{attribute 'GeneratedUsingTerminal: EL5112-0000-0016'}
{attribute addProperty BoxType "EL5112-0000-0016"}
{attribute addProperty Description "EL5112 2Ch. Inc. Encoder 5V (2xAB or 1xABC RS422,TTL)"}
{attribute addProperty Physics "KK"}
{attribute addProperty Id "ENC_Status_Channel_1AT %I*ENC_Status_Channel_10A67E5232ENC_Control_Channel_1AT %Q*ENC_Control_Channel_4C8A739514WcStateAT %I*WcState_9091E0EB2InfoDataAT %I*InfoData_32EB74EA10"}
{attribute addProperty CRC "2247317062"}
{attribute addProperty Size "58"}
TYPE EL5112_85F35646 EXTENDS EtcSlaveTerminalBase_947E5A46 :
STRUCT
	{attribute addProperty Name "ENC_Status_Channel_1"}
	ENC_Status_Channel_1 : ENC_Status_Channel_10A67E52;
	{attribute addProperty Name "ENC_Control_Channel_1"}
	ENC_Control_Channel_1 : ENC_Control_Channel_4C8A7395;
	{attribute addProperty Name "WcState"}
	WcState : WcState_9091E0EB;
	{attribute addProperty Name "InfoData"}
	InfoData : InfoData_32EB74EA;
END_STRUCT
END_TYPE

(* stored: Version 1.2.0.0, ProductVersion 3.1.4024.9
   DUT EL5112_85F35646: Id {9885327f-f7eb-4207-8e2f-76aa33c4e700} *)
